(* IEC 61131-3 sources: git_feedingMachine/lib/test, 2 files *)

(* ---- testTank.st ---- *)
USING AxUnit;
USING TankLib;

NAMESPACE Mytest_Tank

    {TestFixture}
    CLASS Tank_Test_Class
        VAR PRIVATE
            t : Tank;
            vin:Valve;
            vout:Valve;
            _outPutSignalIn : BOOL;
            _outPutSignalOut : BOOL;
        END_VAR

        {Test}
        METHOD PUBLIC Test_FillingMethod_Expect_vin_Open_vout_Closed
            t.Init(vin,vout);
            t.Filling();
            vin.WriteCyclic(outPutSignal => _outPutSignalIn);
            vout.WriteCyclic(outPutSignal => _outPutSignalOut);
            AxUnit.Assert.Equal(actual := _outPutSignalIn, expected := TRUE);
            AxUnit.Assert.Equal(actual := _outPutSignalOut, expected := FALSE);
            ;
        END_METHOD

        {Test}
        METHOD PUBLIC Test_FlushingMethod_Expect_vin_Open_vout_Open
            t.Init(vin,vout);
            t.Flushing();
            vin.WriteCyclic(outPutSignal => _outPutSignalIn);
            vout.WriteCyclic(outPutSignal => _outPutSignalOut);
            AxUnit.Assert.Equal(actual := _outPutSignalIn, expected := TRUE);
            AxUnit.Assert.Equal(actual := _outPutSignalOut, expected := TRUE);
            ;
        END_METHOD

        {Test}
        METHOD PUBLIC Test_CloseMethod_Expect_vin_Closed_vout_Closed
            t.Init(vin,vout);
            t.Close();
            vin.WriteCyclic(outPutSignal => _outPutSignalIn);
            vout.WriteCyclic(outPutSignal => _outPutSignalOut);
            AxUnit.Assert.Equal(actual := _outPutSignalIn, expected := FALSE);
            AxUnit.Assert.Equal(actual := _outPutSignalOut, expected := FALSE);
            ;
        END_METHOD

        {Test}
        METHOD PUBLIC Test_FeedingMethod_Expect_vin_Closed_vout_Open
            t.Init(vin,vout);
            t.Feeding();
            vin.WriteCyclic(outPutSignal => _outPutSignalIn);
            vout.WriteCyclic(outPutSignal => _outPutSignalOut);
            AxUnit.Assert.Equal(actual := _outPutSignalIn, expected := FALSE);
            AxUnit.Assert.Equal(actual := _outPutSignalOut, expected := TRUE);
            ;
        END_METHOD

    END_CLASS

END_NAMESPACE

(* ---- testValve.st ---- *)
USING UserAsserts;
USING AxUnit;
USING TankLib;
NAMESPACE Mytest_Valve
    {TestFixture}
    CLASS Valve_Test_Class
        VAR
            v : Valve;
            vout : BOOL;
        END_VAR

        {Test}
        METHOD PUBLIC Testvout_default_value_expect_false
            v.Close();
            v.WriteCyclic(outPutSignal => vout);
            AxUnit.Assert.Equal(expected := FALSE, actual := vout);
        END_METHOD

        {Test}
        METHOD PUBLIC Test_ValveClose_default_value_expect_false
            v.Open();
            v.Close();
            v.WriteCyclic(outPutSignal => vout);
            AxUnit.Assert.Equal(expected := FALSE, actual := vout);
        END_METHOD

        {Test}
        METHOD PUBLIC Test1
            VAR_TEMP
                result:BOOL;
            END_VAR
            v.Open();
            v.WriteCyclic(outPutSignal => result);
            AxUnit.Assert.Equal(expected := TRUE,actual := result);
        END_METHOD

        {Test}
        METHOD PUBLIC Test_GetStateOf_ClosedValve
            AxUnit.Assert.Equal(TRUE, Equal(ValveState#Closed,v.GetState()) );
        END_METHOD

        {Test}
        METHOD PUBLIC Test_GetStateOf_OpenedValve
            v.Open();
            AxUnit.Assert.Equal(TRUE, Equal(ValveState#Opened,v.GetState()) );
        END_METHOD

    END_CLASS
END_NAMESPACE
